// Mitsubishi GX Works2 project: Project 1.2   PLC: Q03UDV

PROGRAM MAIN
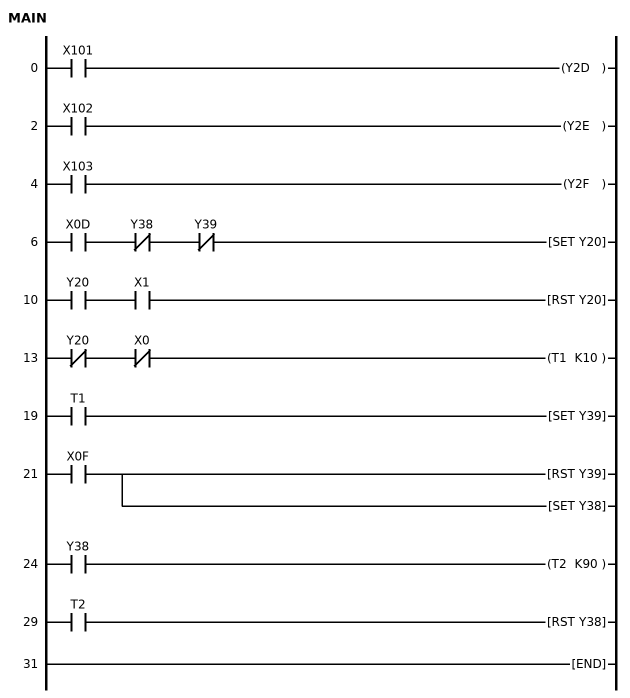
0     LD      X101
      OUT     Y2D
2     LD      X102
      OUT     Y2E
4     LD      X103
      OUT     Y2F
6     LD      X0D
      ANI     Y38
      ANI     Y39
      SET     Y20
10    LD      Y20
      AND     X1
      RST     Y20
13    LDI     Y20
      ANI     X0
      OUT     T1 K10
19    LD      T1
      SET     Y39
21    LD      X0F
      RST     Y39
      SET     Y38
24    LD      Y38
      OUT     T2 K90
29    LD      T2
      RST     Y38
31    END
END_PROGRAM

// device comments not shown above
X110  ; A Supply Switch
X120  ; B Supply Switch
X210  ; Motor Forward
X220  ; Motor Backward
